DATA_BLOCK "ST10_CountCycleTimeMain_DB"
{ S7_Optimized_Access := 'TRUE' }
VERSION : 0.1
NON_RETAIN
"ST10_CountCycleTimeMain"

BEGIN

END_DATA_BLOCK

